FUNCTION_BLOCK AxisPower EXTENDS TaskBase
VAR
	mcPower : Tc2_MC2.MC_Power;
	AxisReference : REFERENCE TO Tc2_MC2.AXIS_REF;
	EnableAxis : BOOL;
END_VAR

METHOD Abort : BOOL
mcPower.Enable := mcPower.Enable_Negative := mcPower.Enable_Positive := FALSE;
_Busy := FALSE;
EnableAxis := FALSE;
Abort := TRUE;
State := 0;
END_METHOD

METHOD Cycle : BOOL
VAR_INPUT
END_VAR
CASE State OF
	0:
		IF EnableAxis THEN
			_Done := FALSE;
			_Error := FALSE;
			_Busy := TRUE;
			mcPower.Enable := mcPower.Enable_Negative := mcPower.Enable_Positive := TRUE;
			mcPower.Override := 100;
			State := 10;
		END_IF
	
	10:
		IF mcPower.Status THEN
			_Busy := FALSE;
			_Done := TRUE;
			State := 20;
		END_IF
	
	20:
		IF NOT EnableAxis THEN
			_Done := FALSE;
			_Busy := TRUE;
			mcPower.Enable := mcPower.Enable_Negative := mcPower.Enable_Positive := FALSE;
			State := 30;
		END_IF
	30:
		IF NOT mcPower.Status THEN
			_Busy := FALSE;
			_Done := TRUE;
			State := 0;
		END_IF
END_CASE

mcPower(Axis := AxisReference);
END_METHOD

METHOD Disable : BOOL
VAR_INPUT
END_VAR
IF NOT EnableAxis THEN
	RETURN;
END_IF
Disable := TRUE;
EnableAxis := FALSE;
END_METHOD

METHOD Enable : BOOL
VAR_INPUT
END_VAR
IF EnableAxis THEN
	RETURN;
END_IF
Enable := EnableAxis := true;
END_METHOD

METHOD FB_init : BOOL
VAR_INPUT
	bInitRetains : BOOL; // if TRUE, the retain variables are initialized (warm start / cold start)
	bInCopyCode : BOOL;  // if TRUE, the instance afterwards gets moved into the copy code (online change)
	axis : reference TO AXIS_REF;
END_VAR
AxisReference REF= axis;
END_METHOD

END_FUNCTION_BLOCK

(* stored: Version 1.1.0.1, ProductVersion 3.1.4024.12
   POU AxisPower: Id {9020922a-7816-4155-9202-ac5854f794ea}, SpecialFunc None
   Method Abort: Id {93bd9e75-34cf-4a99-8cdf-c273723a870d}
   Method Cycle: Id {c1cf1940-bcdc-4ac4-844e-317c1f14fe0e}
   Method Disable: Id {0a54e8c6-7456-4747-8eeb-b97b9078e709}
   Method Enable: Id {afe5d65c-4532-4d19-b244-08cfed3445ed}
   Method FB_init: Id {03d72923-bd2d-4684-847b-d6b404bc945a} *)
